Fanuc KAREL source: IO0034.KL

-- PROVISIONAL review KL for V1013-1; original PC SHA256 d79c29b1997b143f7a1c44f41a85a1aeaf157f4dc4545dc842ed4705a795aea3
-- Incomplete behavior may be omitted. Consult companion uncertainty JSON. Do not deploy.
PROGRAM IO0034
%NOLOCKGROUP
-- UNRESOLVED_LOCAL_POOL 5 cells at code offset 13; source declarations unknown
-- DIRECT_LOCAL_WORD_ACCESS alone does not prove INTEGER, REAL, or BOOLEAN
BEGIN
  -- UNRESOLVED_PC offsets 0-18; opcodes 2B,2C,7B
  -- UNRESOLVED_PC offsets 23-30; opcodes 9D,23
  -- UNRESOLVED_PC offsets 35-49; opcodes 2E,22,9D,33,35
  -- UNRESOLVED_PC offsets 54-61; opcodes 9D,23
  -- UNRESOLVED_PC offsets 66-77; opcodes 2E,23
  -- UNRESOLVED_PC offsets 82-104; opcodes 21,22,21,33,34,1A
  -- UNRESOLVED_PC offsets 109-113; opcodes 7F
  -- UNRESOLVED_PC offsets 118-122; opcodes 27,AA
  -- UNRESOLVED_PC offsets 127-131; opcodes 7F
END IO0034
